Yaskawa INFORM job: R1_W63-A1(120,-90)KM-OK_R2.JBI

/JOB
//NAME R1_W63-A1(120,-90)KM-OK_R2
///FOLDERNAME KRIS-SCIANA
//POS
///NPOS 37,37,0,3,0,0
///TOOL 0
///POSTYPE PULSE
///PULSE
C00000=-6494,-75728,-88783,9927,90662,-21871
C00001=-76570,-4200,-56852,-3495,80469,-6039
C00002=-120300,77172,47502,-18765,68874,11972
C00003=-132514,56441,47332,-3289,65899,22293
C00004=-133277,63718,58812,-3130,62549,22103
C00005=-133575,67040,63977,-3074,61067,22030
C00006=-133575,68098,66659,-3107,59964,22061
C00007=-133575,67040,63977,-3074,61067,22030
C00008=-133575,67040,63977,-3074,61067,22030
C00009=-133450,70639,68253,-3139,60291,22100
C00010=-134019,69654,66695,-2935,60722,21870
C00011=-134655,65869,63126,-2717,60950,21621
C00012=-135298,66430,63779,-2505,60812,21379
C00013=-134655,65869,63126,-2717,60950,21621
C00014=-134364,62559,57990,-2776,62418,21696
C00015=-133617,55287,46555,-2941,65742,21892
C00016=-112115,61855,50901,4001,73980,8160
C00017=-112331,73122,68555,4159,68928,7910
C00018=-112350,74742,71432,4189,67993,7872
C00019=-112346,74422,70868,4183,68175,7879
C00020=-112381,75999,72649,4200,67892,7857
C00021=-112299,71765,67058,4149,69149,7930
C00022=-114491,51106,36872,4426,77207,7440
C00023=-160530,30370,22657,949,47620,-12111
C00024=-160530,30370,22657,949,47620,-12111
C00025=-153919,83642,85160,-11029,55472,-9179
C00026=-157150,45041,48687,15575,47374,-13815
C00027=-157183,45552,50297,15775,46678,-13949
C00028=-156744,89080,88941,7300,63205,-11720
C00029=-141018,57292,50426,3243,69519,-5670
C00030=-128529,48357,40466,187,70792,-1190
C00031=-140701,60474,59315,29933,72810,-5893
C00032=-148105,52207,40176,29980,82020,-6383
C00033=-135666,25352,5121,11647,67948,-24320
C00034=-135594,26700,-8269,11068,76272,-23437
C00035=-135685,26741,-8205,11256,29920,-23439
C00036=-1222,-82811,-95096,11256,91671,-23439
BC00000=124218,683035,1059245
BC00001=211926,717459,1063229
BC00002=311705,756620,1067762
BC00003=311879,816330,1067608
BC00004=311879,816330,1067608
BC00005=311879,816330,1067608
BC00006=311879,816330,1067608
BC00007=311879,816330,1067608
BC00008=311879,816330,1067608
BC00009=311879,816330,1067608
BC00010=311879,816330,1067608
BC00011=311879,816330,1067608
BC00012=311879,816330,1067608
BC00013=311879,816330,1067608
BC00014=311879,816330,1067608
BC00015=311879,816330,1067608
BC00016=323115,818777,1066878
BC00017=323115,818777,1066878
BC00018=323115,818777,1066878
BC00019=323115,818777,1066878
BC00020=323115,818777,1066878
BC00021=323115,818777,1066878
BC00022=323115,818777,1066878
BC00023=394257,833547,1058815
BC00024=394257,833547,1058815
BC00025=394257,833547,1058815
BC00026=394257,833522,1068222
BC00027=394257,833522,1068222
BC00028=394257,833547,1058815
BC00029=394257,833547,1058815
BC00030=394257,833547,1058815
BC00031=394257,833547,1058815
BC00032=394257,833547,1058815
BC00033=394257,833546,1058813
BC00034=394171,833543,1058850
BC00035=346692,691893,1058850
BC00036=115533,679626,1058850
///POSTYPE BASE
///RECTAN
///RCONF 0,0,0,0,0,0,0,0,0,0,0,0,0,0,0,0,0,0,0,0,0,0,0,0
P00006=0.222,-3.123,-1.508,0.0000,0.0000,0.0000
P00021=-0.225,-6.128,-0.405,0.0000,0.0000,0.0000
P00022=0.222,-3.123,-1.508,0.0000,0.0000,0.0000
//INST
///DATE 2024/07/25 17:47
///ATTR SC,RW
///GROUP1 RB1,BS1
NOP
'Path S1152
SFTOF
MOVJ C00000 BC00000 VJ=50.00
MOVJ C00001 BC00001 VJ=50.00
MOVJ C00002 BC00002 VJ=20.00
MOVJ C00003 BC00003 VJ=20.00
MOVL C00004 BC00004 V=100.0
MOVL C00005 BC00005 V=60.0
REFP 3 C00006 BC00006
CALL JOB:SEARCH-R1
SET P021 P006
SFTON P021
MOVL C00007 BC00007 V=60.0
MOVL C00008 BC00008 V=60.0
REFP 3 C00009 BC00009
CALL JOB:SEARCH-R1
SET P021 P006
SFTON P021
MOVL C00010 BC00010 V=60.0
MOVL C00011 BC00011 V=60.0
REFP 3 C00012 BC00012
CALL JOB:SEARCH-R1
SET P021 P006
SFTON P021
MOVL C00013 BC00013 V=60.0
MOVL C00014 BC00014 V=100.0
MOVL C00015 BC00015 V=100.0
'Path S1153
SFTOF
MOVJ C00016 BC00016 VJ=20.00
MOVL C00017 BC00017 V=100.0
REFP 3 C00018 BC00018
CALL JOB:SEARCH-R1
SET P022 P006
SFTON P022
MOVL C00019 BC00019 V=60.0
REFP 3 C00020 BC00020
CALL JOB:SEARCH-R1
SET P022 P006
SFTON P022
MOVL C00021 BC00021 V=60.0
MOVL C00022 BC00022 V=100.0
'Path W1154
SFTOF
SFTON P021
MOVJ C00023 BC00023 VJ=20.00
MOVL C00024 BC00024 V=100.0
MOVL C00025 BC00025 V=100.0 PL=0
REFP 1 C00026 BC00026
REFP 2 C00027 BC00027
MACRO1 MJ#(0) ARGF9
ARCON
MOVL C00028 BC00028 V=11.2
SFTON P022
MOVL C00029 BC00029 V=11.2
MOVL C00030 BC00030 V=11.2
MOVL C00031 BC00031 V=10.8
ARCOF
MOVL C00032 BC00032 V=100.0
MOVL C00033 BC00033 V=200.0
SFTOF
MOVJ C00034 BC00034 VJ=20.00
MOVJ C00035 BC00035 VJ=20.00
MOVJ C00036 BC00036 VJ=100.00
SFTOF
END
